ABB RobotStudio station: Solution5_20230425-115824.rsstn

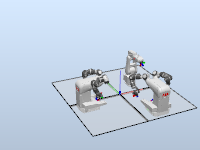
Station Solution5 (saved by RobotStudio 21.4.9700.0)
Controller Yumi, task T_ROB_L: task frame (RAPID world) sits at (-500, -35, 0) mm in the station
Controller Yumi, task T_ROB_R: task frame (RAPID world) sits at (-500, -35, 0) mm in the station
Controller IRB120_3_58, task T_ROB1: task frame (RAPID world) sits at (400, 300, 0) mm, rotated rx 0 ry 0 rz -90 deg in the station
Controller IRB14000, task T_ROB_L: task frame (RAPID world) sits at (400, -500, 0) mm, rotated rx 0 ry 0 rz 90 deg in the station
Controller IRB14000, task T_ROB_R: task frame (RAPID world) sits at (400, -500, 0) mm, rotated rx 0 ry 0 rz 90 deg in the station
Controller IRB14000
  mechanical unit ROB_R: IRB14000_0.5_0.5_R, 6 joints, base frame (0, 0, 0) mm
  mechanical unit ROB_R_7: IRB14000_0.5_0.5_R, 1 joints, base frame (0, 0, 0) mm
  mechanical unit ROB_L: IRB14000_0.5_0.5_L, 6 joints, base frame (0, 0, 0) mm
  mechanical unit ROB_L_7: IRB14000_0.5_0.5_L, 1 joints, base frame (0, 0, 0) mm
Controller IRB120_3_58
  mechanical unit ROB_1: IRB120_demo, 6 joints, base frame (0, 0, 0) mm
Controller Yumi
  mechanical unit ROB_R: IRB14000_0.5_0.5_R_2, 6 joints, base frame (0, 0, 0) mm
  mechanical unit ROB_R_7: IRB14000_0.5_0.5_R_2, 1 joints, base frame (0, 0, 0) mm
  mechanical unit ROB_L: IRB14000_0.5_0.5_L_2, 6 joints, base frame (0, 0, 0) mm
  mechanical unit ROB_L_7: IRB14000_0.5_0.5_L_2, 1 joints, base frame (0, 0, 0) mm
Layout (positions relative to the parent item):
  - yumi_demo [mechanism, from Robots\IRB14000_0.5_0.5__01.rslib] at (400, -500, 0) mm, rotated rx 0 ry 0 rz 90 deg
  - IRB14000_0.5_0.5_R [mechanism, from Robots\IRB14000_0.5_0.5__01.rslib] at (400, -500, 0) mm, rotated rx 0 ry 0 rz 90 deg; joint values [0, -2.2689, -2.3562, 0.5236, 0, 0.6981, 0] (rad or m)
  - IRB14000_0.5_0.5_L [mechanism, from Robots\IRB14000_0.5_0.5__01.rslib] at (400, -500, 0) mm, rotated rx 0 ry 0 rz 90 deg; joint values [1.3562, 0.5925, 0.0328, 0.5875, -1.9784, 1.0159, -1.5366] (rad or m)
  - IRB120_demo [mechanism, from Robots\IRB120_3_58_G_01.rslib] at (400, 300, 0) mm, rotated rx 0 ry 0 rz -90 deg; joint values [0, 0, 0, 0, 0.5236, 0] (rad or m)
  - IRB14000_0.5_0.5 [mechanism, from Robots\IRB14000_0.5_0.5__01.rslib] at (-500, -35, 0) mm
  - IRB14000_0.5_0.5_R_2 [mechanism, from Robots\IRB14000_0.5_0.5__01.rslib] at (-500, -35, 0) mm; joint values [0, -2.2689, -2.3562, 0.5236, 0, 0.6981, 0] (rad or m)
  - IRB14000_0.5_0.5_L_2 [mechanism, from Robots\IRB14000_0.5_0.5__01.rslib] at (-500, -35, 0) mm; joint values [0, -2.2689, 2.3562, 0.5236, 0, 0.6981, 0] (rad or m)
